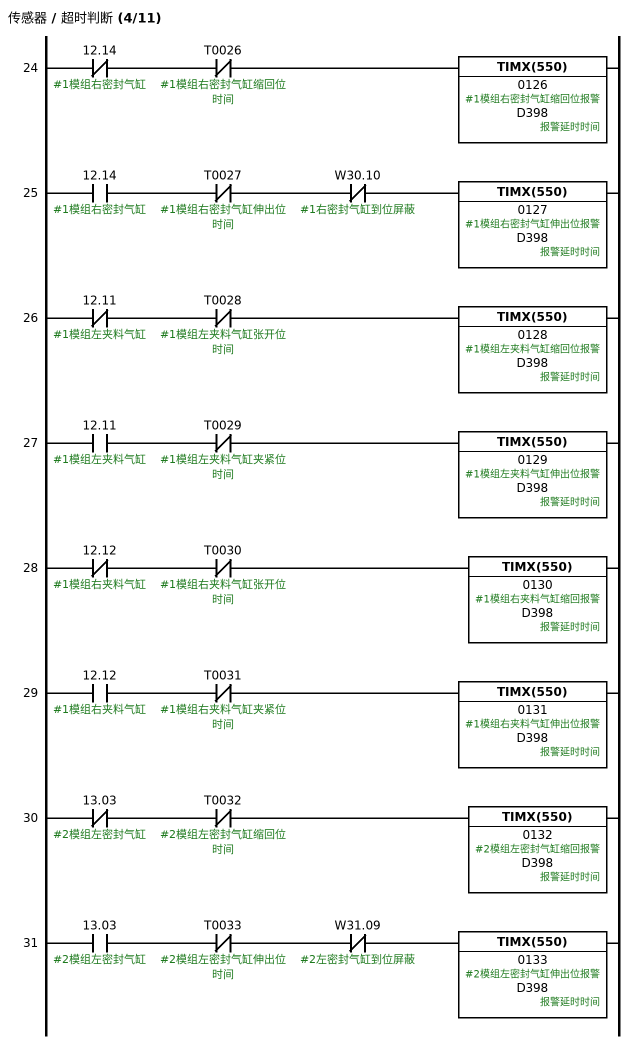
; [picture p65: 传感器 / 超时判断, rungs 24-31]
; rung 24
LDNOT 12.14  ; #1模组右密封气缸
ANDNOT T0026  ; #1模组右密封气缸缩回位时间
TIMX(550) 0126 D398  ; 报警延时时间, #1模组右密封气缸缩回位报警
; rung 25
LD 12.14  ; #1模组右密封气缸
ANDNOT T0027  ; #1模组右密封气缸伸出位时间
ANDNOT W30.10  ; #1右密封气缸到位屏蔽
TIMX(550) 0127 D398  ; 报警延时时间, #1模组右密封气缸伸出位报警
; rung 26
LDNOT 12.11  ; #1模组左夹料气缸
ANDNOT T0028  ; #1模组左夹料气缸张开位时间
TIMX(550) 0128 D398  ; 报警延时时间, #1模组左夹料气缸缩回位报警
; rung 27
LD 12.11  ; #1模组左夹料气缸
ANDNOT T0029  ; #1模组左夹料气缸夹紧位时间
TIMX(550) 0129 D398  ; 报警延时时间, #1模组左夹料气缸伸出位报警
; rung 28
LDNOT 12.12  ; #1模组右夹料气缸
ANDNOT T0030  ; #1模组右夹料气缸张开位时间
TIMX(550) 0130 D398  ; 报警延时时间, #1模组右夹料气缸缩回报警
; rung 29
LD 12.12  ; #1模组右夹料气缸
ANDNOT T0031  ; #1模组右夹料气缸夹紧位时间
TIMX(550) 0131 D398  ; 报警延时时间, #1模组右夹料气缸伸出位报警
; rung 30
LDNOT 13.03  ; #2模组左密封气缸
ANDNOT T0032  ; #2模组左密封气缸缩回位时间
TIMX(550) 0132 D398  ; 报警延时时间, #2模组左密封气缸缩回报警
; rung 31
LD 13.03  ; #2模组左密封气缸
ANDNOT T0033  ; #2模组左密封气缸伸出位时间
ANDNOT W31.09  ; #2左密封气缸到位屏蔽
TIMX(550) 0133 D398  ; 报警延时时间, #2模组左密封气缸伸出位报警

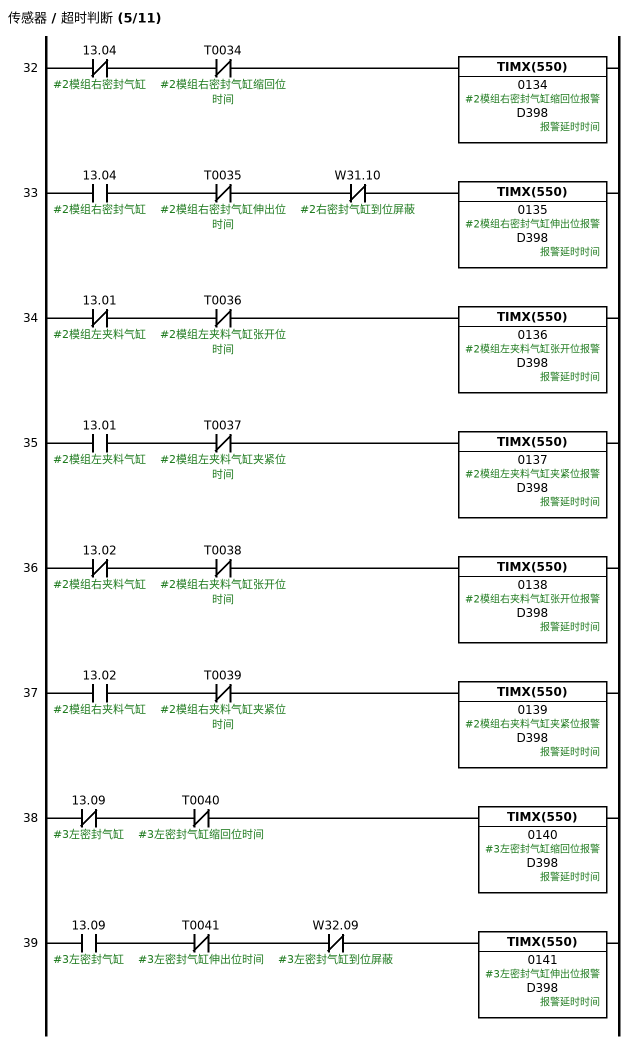
; rung 32
LDNOT 13.04  ; #2模组右密封气缸
ANDNOT T0034  ; #2模组右密封气缸缩回位时间
TIMX(550) 0134 D398  ; 报警延时时间, #2模组右密封气缸缩回位报警
; rung 33
LD 13.04  ; #2模组右密封气缸
ANDNOT T0035  ; #2模组右密封气缸伸出位时间
ANDNOT W31.10  ; #2右密封气缸到位屏蔽
TIMX(550) 0135 D398  ; 报警延时时间, #2模组右密封气缸伸出位报警
; rung 34
LDNOT 13.01  ; #2模组左夹料气缸
ANDNOT T0036  ; #2模组左夹料气缸张开位时间
TIMX(550) 0136 D398  ; 报警延时时间, #2模组左夹料气缸张开位报警
; rung 35
LD 13.01  ; #2模组左夹料气缸
ANDNOT T0037  ; #2模组左夹料气缸夹紧位时间
TIMX(550) 0137 D398  ; 报警延时时间, #2模组左夹料气缸夹紧位报警
; rung 36
LDNOT 13.02  ; #2模组右夹料气缸
ANDNOT T0038  ; #2模组右夹料气缸张开位时间
TIMX(550) 0138 D398  ; 报警延时时间, #2模组右夹料气缸张开位报警
; rung 37
LD 13.02  ; #2模组右夹料气缸
ANDNOT T0039  ; #2模组右夹料气缸夹紧位时间
TIMX(550) 0139 D398  ; 报警延时时间, #2模组右夹料气缸夹紧位报警
; rung 38
LDNOT 13.09  ; #3左密封气缸
ANDNOT T0040  ; #3左密封气缸缩回位时间
TIMX(550) 0140 D398  ; 报警延时时间, #3左密封气缸缩回位报警
; rung 39
LD 13.09  ; #3左密封气缸
ANDNOT T0041  ; #3左密封气缸伸出位时间
ANDNOT W32.09  ; #3左密封气缸到位屏蔽
TIMX(550) 0141 D398  ; 报警延时时间, #3左密封气缸伸出位报警

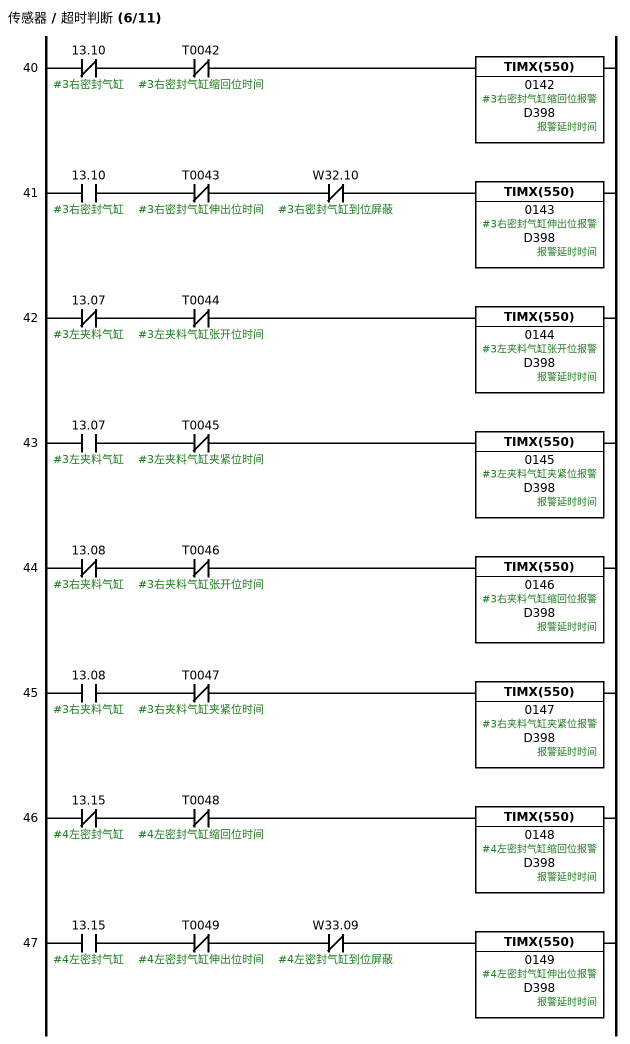
; rung 40
LDNOT 13.10  ; #3右密封气缸
ANDNOT T0042  ; #3右密封气缸缩回位时间
TIMX(550) 0142 D398  ; 报警延时时间, #3右密封气缸缩回位报警
; rung 41
LD 13.10  ; #3右密封气缸
ANDNOT T0043  ; #3右密封气缸伸出位时间
ANDNOT W32.10  ; #3右密封气缸到位屏蔽
TIMX(550) 0143 D398  ; 报警延时时间, #3右密封气缸伸出位报警
; rung 42
LDNOT 13.07  ; #3左夹料气缸
ANDNOT T0044  ; #3左夹料气缸张开位时间
TIMX(550) 0144 D398  ; 报警延时时间, #3左夹料气缸张开位报警
; rung 43
LD 13.07  ; #3左夹料气缸
ANDNOT T0045  ; #3左夹料气缸夹紧位时间
TIMX(550) 0145 D398  ; 报警延时时间, #3左夹料气缸夹紧位报警
; rung 44
LDNOT 13.08  ; #3右夹料气缸
ANDNOT T0046  ; #3右夹料气缸张开位时间
TIMX(550) 0146 D398  ; 报警延时时间, #3右夹料气缸缩回位报警
; rung 45
LD 13.08  ; #3右夹料气缸
ANDNOT T0047  ; #3右夹料气缸夹紧位时间
TIMX(550) 0147 D398  ; 报警延时时间, #3右夹料气缸夹紧位报警
; rung 46
LDNOT 13.15  ; #4左密封气缸
ANDNOT T0048  ; #4左密封气缸缩回位时间
TIMX(550) 0148 D398  ; 报警延时时间, #4左密封气缸缩回位报警
; rung 47
LD 13.15  ; #4左密封气缸
ANDNOT T0049  ; #4左密封气缸伸出位时间
ANDNOT W33.09  ; #4左密封气缸到位屏蔽
TIMX(550) 0149 D398  ; 报警延时时间, #4左密封气缸伸出位报警

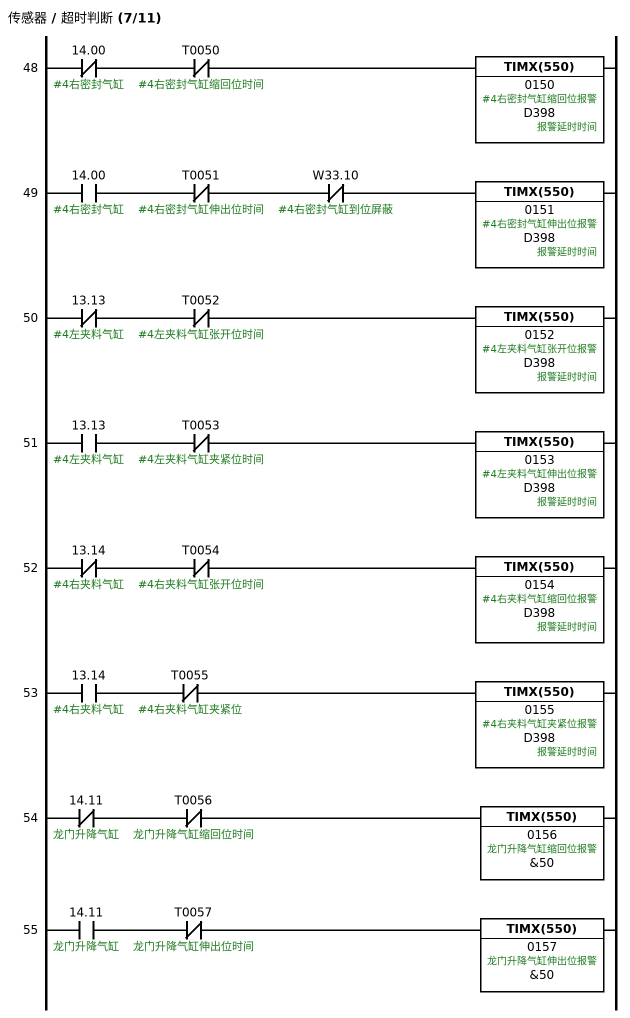
; rung 48
LDNOT 14.00  ; #4右密封气缸
ANDNOT T0050  ; #4右密封气缸缩回位时间
TIMX(550) 0150 D398  ; 报警延时时间, #4右密封气缸缩回位报警
; rung 49
LD 14.00  ; #4右密封气缸
ANDNOT T0051  ; #4右密封气缸伸出位时间
ANDNOT W33.10  ; #4右密封气缸到位屏蔽
TIMX(550) 0151 D398  ; 报警延时时间, #4右密封气缸伸出位报警
; rung 50
LDNOT 13.13  ; #4左夹料气缸
ANDNOT T0052  ; #4左夹料气缸张开位时间
TIMX(550) 0152 D398  ; 报警延时时间, #4左夹料气缸张开位报警
; rung 51
LD 13.13  ; #4左夹料气缸
ANDNOT T0053  ; #4左夹料气缸夹紧位时间
TIMX(550) 0153 D398  ; 报警延时时间, #4左夹料气缸伸出位报警
; rung 52
LDNOT 13.14  ; #4右夹料气缸
ANDNOT T0054  ; #4右夹料气缸张开位时间
TIMX(550) 0154 D398  ; 报警延时时间, #4右夹料气缸缩回位报警
; rung 53
LD 13.14  ; #4右夹料气缸
ANDNOT T0055  ; #4右夹料气缸夹紧位
TIMX(550) 0155 D398  ; 报警延时时间, #4右夹料气缸夹紧位报警
; rung 54
LDNOT 14.11  ; 龙门升降气缸
ANDNOT T0056  ; 龙门升降气缸缩回位时间
TIMX(550) 0156 &50  ; 龙门升降气缸缩回位报警
; rung 55
LD 14.11  ; 龙门升降气缸
ANDNOT T0057  ; 龙门升降气缸伸出位时间
TIMX(550) 0157 &50  ; 龙门升降气缸伸出位报警

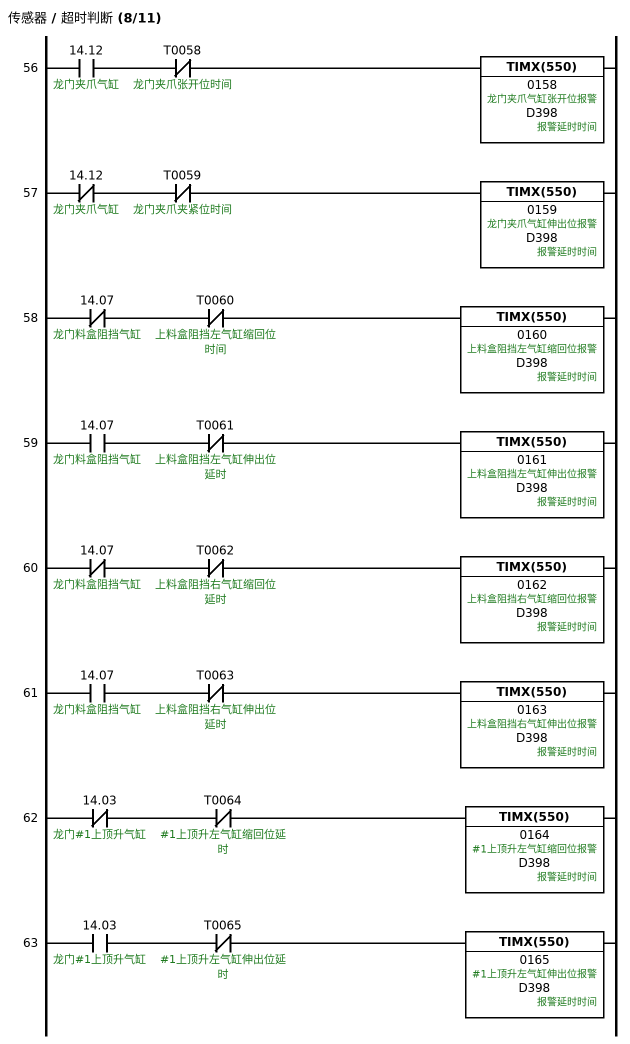
; rung 56
LD 14.12  ; 龙门夹爪气缸
ANDNOT T0058  ; 龙门夹爪张开位时间
TIMX(550) 0158 D398  ; 报警延时时间, 龙门夹爪气缸张开位报警
; rung 57
LDNOT 14.12  ; 龙门夹爪气缸
ANDNOT T0059  ; 龙门夹爪夹紧位时间
TIMX(550) 0159 D398  ; 报警延时时间, 龙门夹爪气缸伸出位报警
; rung 58
LDNOT 14.07  ; 龙门料盒阻挡气缸
ANDNOT T0060  ; 上料盒阻挡左气缸缩回位时间
TIMX(550) 0160 D398  ; 报警延时时间, 上料盒阻挡左气缸缩回位报警
; rung 59
LD 14.07  ; 龙门料盒阻挡气缸
ANDNOT T0061  ; 上料盒阻挡左气缸伸出位延时
TIMX(550) 0161 D398  ; 报警延时时间, 上料盒阻挡左气缸伸出位报警
; rung 60
LDNOT 14.07  ; 龙门料盒阻挡气缸
ANDNOT T0062  ; 上料盒阻挡右气缸缩回位延时
TIMX(550) 0162 D398  ; 报警延时时间, 上料盒阻挡右气缸缩回位报警
; rung 61
LD 14.07  ; 龙门料盒阻挡气缸
ANDNOT T0063  ; 上料盒阻挡右气缸伸出位延时
TIMX(550) 0163 D398  ; 报警延时时间, 上料盒阻挡右气缸伸出位报警
; rung 62
LDNOT 14.03  ; 龙门#1上顶升气缸
ANDNOT T0064  ; #1上顶升左气缸缩回位延时
TIMX(550) 0164 D398  ; 报警延时时间, #1上顶升左气缸缩回位报警
; rung 63
LD 14.03  ; 龙门#1上顶升气缸
ANDNOT T0065  ; #1上顶升左气缸伸出位延时
TIMX(550) 0165 D398  ; 报警延时时间, #1上顶升左气缸伸出位报警

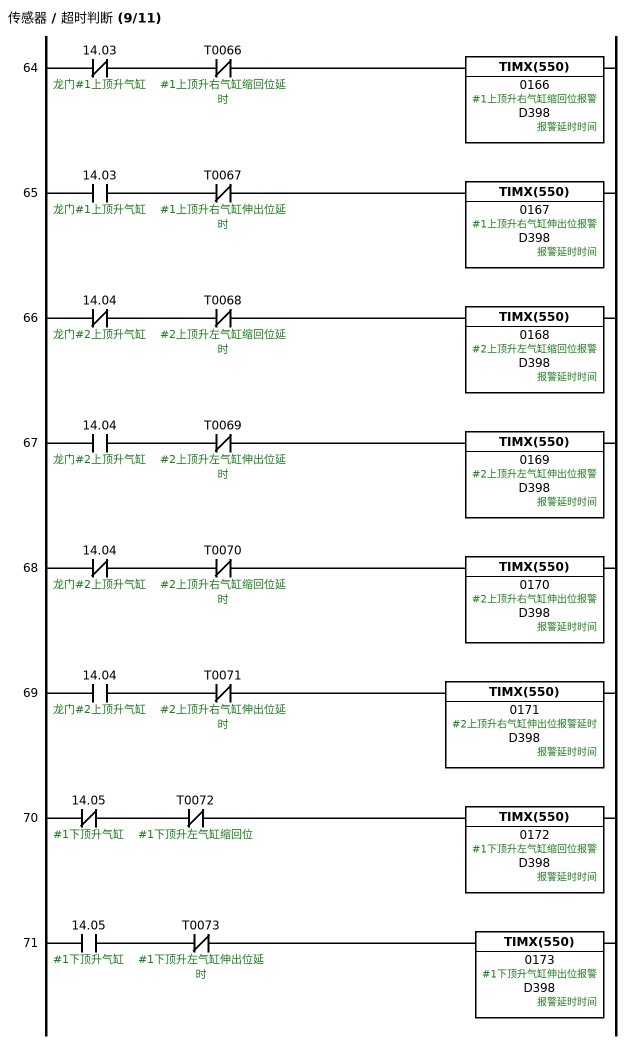
; rung 64
LDNOT 14.03  ; 龙门#1上顶升气缸
ANDNOT T0066  ; #1上顶升右气缸缩回位延时
TIMX(550) 0166 D398  ; 报警延时时间, #1上顶升右气缸缩回位报警
; rung 65
LD 14.03  ; 龙门#1上顶升气缸
ANDNOT T0067  ; #1上顶升右气缸伸出位延时
TIMX(550) 0167 D398  ; 报警延时时间, #1上顶升右气缸伸出位报警
; rung 66
LDNOT 14.04  ; 龙门#2上顶升气缸
ANDNOT T0068  ; #2上顶升左气缸缩回位延时
TIMX(550) 0168 D398  ; 报警延时时间, #2上顶升左气缸缩回位报警
; rung 67
LD 14.04  ; 龙门#2上顶升气缸
ANDNOT T0069  ; #2上顶升左气缸伸出位延时
TIMX(550) 0169 D398  ; 报警延时时间, #2上顶升左气缸伸出位报警
; rung 68
LDNOT 14.04  ; 龙门#2上顶升气缸
ANDNOT T0070  ; #2上顶升右气缸缩回位延时
TIMX(550) 0170 D398  ; 报警延时时间, #2上顶升右气缸伸出位报警
; rung 69
LD 14.04  ; 龙门#2上顶升气缸
ANDNOT T0071  ; #2上顶升右气缸伸出位延时
TIMX(550) 0171 D398  ; 报警延时时间, #2上顶升右气缸伸出位报警延时
; rung 70
LDNOT 14.05  ; #1下顶升气缸
ANDNOT T0072  ; #1下顶升左气缸缩回位
TIMX(550) 0172 D398  ; 报警延时时间, #1下顶升左气缸缩回位报警
; rung 71
LD 14.05  ; #1下顶升气缸
ANDNOT T0073  ; #1下顶升左气缸伸出位延时
TIMX(550) 0173 D398  ; 报警延时时间, #1下顶升气缸伸出位报警

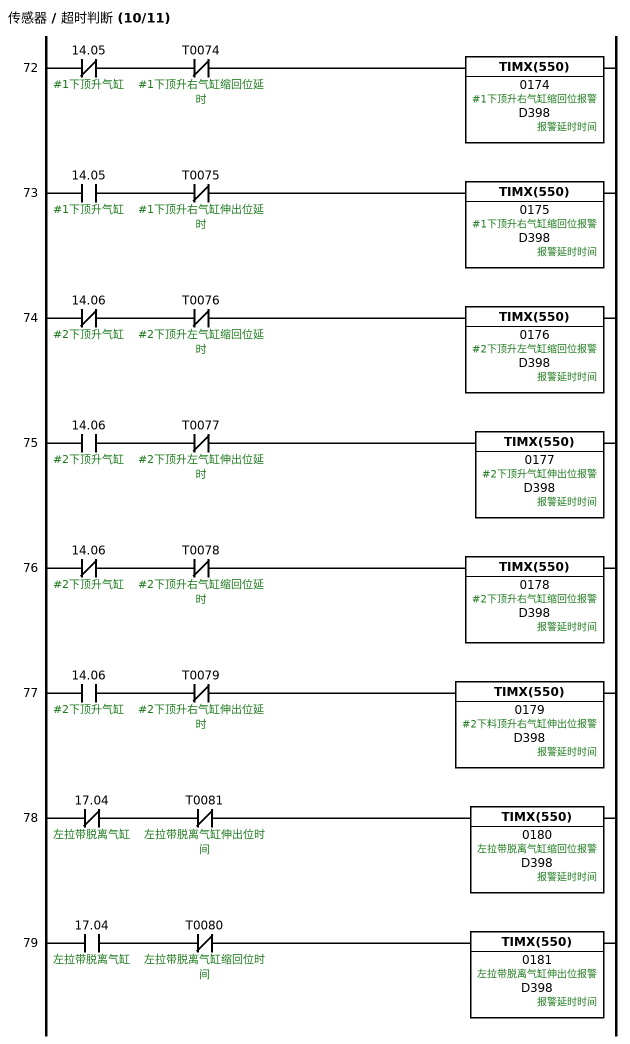
; rung 72
LDNOT 14.05  ; #1下顶升气缸
ANDNOT T0074  ; #1下顶升右气缸缩回位延时
TIMX(550) 0174 D398  ; 报警延时时间, #1下顶升右气缸缩回位报警
; rung 73
LD 14.05  ; #1下顶升气缸
ANDNOT T0075  ; #1下顶升右气缸伸出位延时
TIMX(550) 0175 D398  ; 报警延时时间, #1下顶升右气缸缩回位报警
; rung 74
LDNOT 14.06  ; #2下顶升气缸
ANDNOT T0076  ; #2下顶升左气缸缩回位延时
TIMX(550) 0176 D398  ; 报警延时时间, #2下顶升左气缸缩回位报警
; rung 75
LD 14.06  ; #2下顶升气缸
ANDNOT T0077  ; #2下顶升左气缸伸出位延时
TIMX(550) 0177 D398  ; 报警延时时间, #2下顶升气缸伸出位报警
; rung 76
LDNOT 14.06  ; #2下顶升气缸
ANDNOT T0078  ; #2下顶升右气缸缩回位延时
TIMX(550) 0178 D398  ; 报警延时时间, #2下顶升右气缸缩回位报警
; rung 77
LD 14.06  ; #2下顶升气缸
ANDNOT T0079  ; #2下顶升右气缸伸出位延时
TIMX(550) 0179 D398  ; 报警延时时间, #2下料顶升右气缸伸出位报警
; rung 78
LDNOT 17.04  ; 左拉带脱离气缸
ANDNOT T0081  ; 左拉带脱离气缸伸出位时间
TIMX(550) 0180 D398  ; 报警延时时间, 左拉带脱离气缸缩回位报警
; rung 79
LD 17.04  ; 左拉带脱离气缸
ANDNOT T0080  ; 左拉带脱离气缸缩回位时间
TIMX(550) 0181 D398  ; 报警延时时间, 左拉带脱离气缸伸出位报警

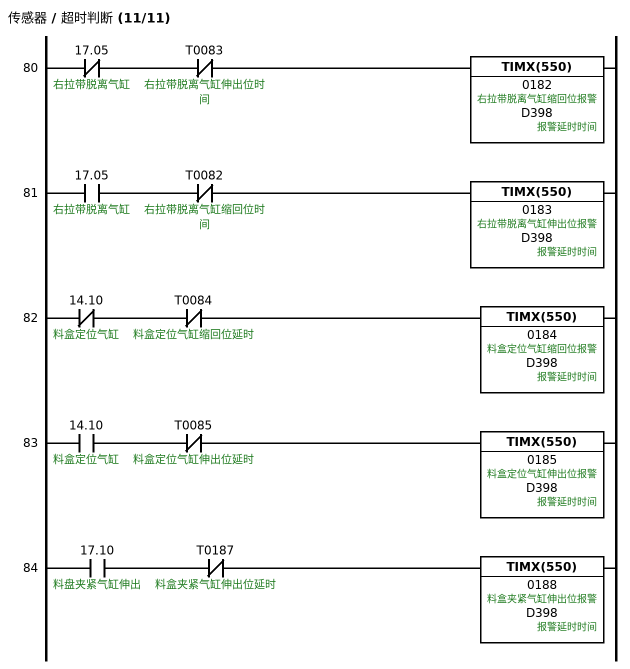
; rung 80
LDNOT 17.05  ; 右拉带脱离气缸
ANDNOT T0083  ; 右拉带脱离气缸伸出位时间
TIMX(550) 0182 D398  ; 报警延时时间, 右拉带脱离气缸缩回位报警
; rung 81
LD 17.05  ; 右拉带脱离气缸
ANDNOT T0082  ; 右拉带脱离气缸缩回位时间
TIMX(550) 0183 D398  ; 报警延时时间, 右拉带脱离气缸伸出位报警
; rung 82
LDNOT 14.10  ; 料盒定位气缸
ANDNOT T0084  ; 料盒定位气缸缩回位延时
TIMX(550) 0184 D398  ; 报警延时时间, 料盒定位气缸缩回位报警
; rung 83
LD 14.10  ; 料盒定位气缸
ANDNOT T0085  ; 料盒定位气缸伸出位延时
TIMX(550) 0185 D398  ; 报警延时时间, 料盒定位气缸伸出位报警
; rung 84
LD 17.10  ; 料盘夹紧气缸伸出
ANDNOT T0187  ; 料盒夹紧气缸伸出位延时
TIMX(550) 0188 D398  ; 报警延时时间, 料盒夹紧气缸伸出位报警

### Section END
; rung 0
END(001)

## Program 上料机构 (cyclic task 2)

### Section 扫码，检测手动

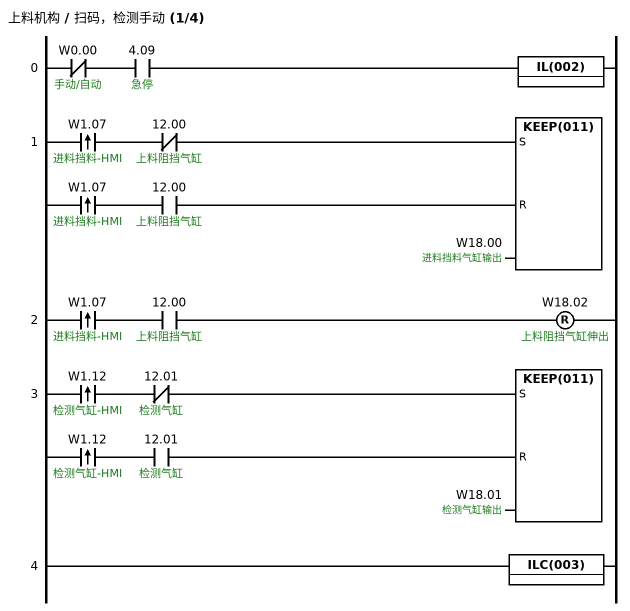
; rung 0
LDNOT W0.00  ; 手动/自动
AND 4.09  ; 急停
IL(002)
; rung 1
@LD W1.07  ; 进料挡料-HMI
ANDNOT 12.00  ; 上料阻挡气缸
@LD W1.07  ; 进料挡料-HMI
AND 12.00  ; 上料阻挡气缸
KEEP(011) W18.00  ; 进料挡料气缸输出
; rung 2
@LD W1.07  ; 进料挡料-HMI
AND 12.00  ; 上料阻挡气缸
RSET W18.02  ; 上料阻挡气缸伸出
; rung 3
@LD W1.12  ; 检测气缸-HMI
ANDNOT 12.01  ; 检测气缸
@LD W1.12  ; 检测气缸-HMI
AND 12.01  ; 检测气缸
KEEP(011) W18.01  ; 检测气缸输出
; rung 4
ILC(003)

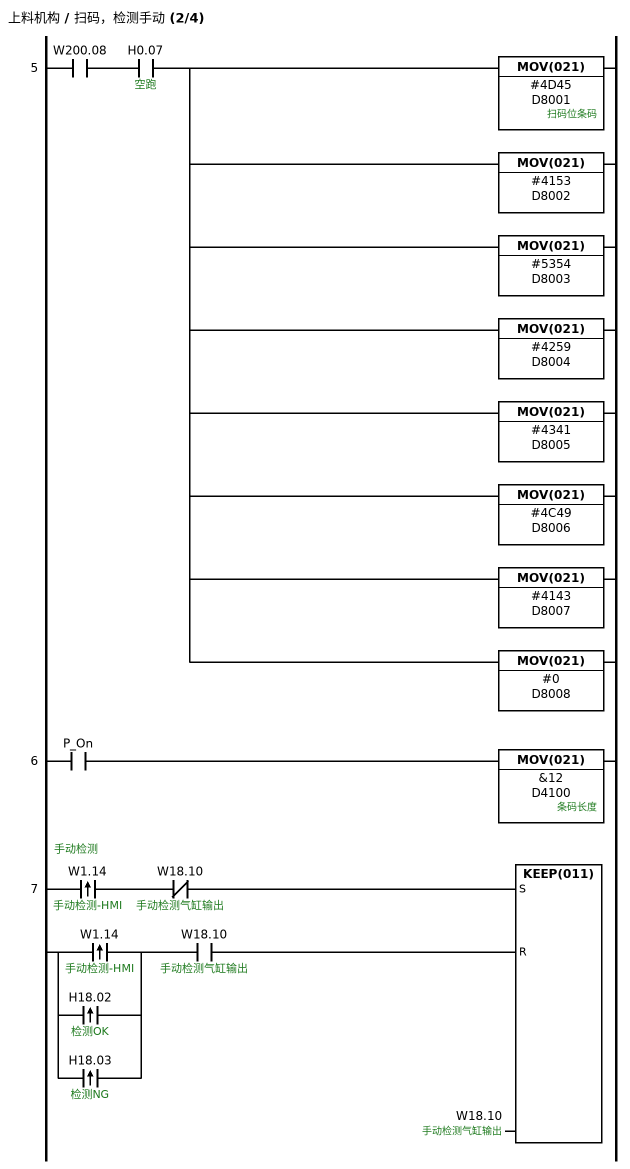
; rung 5
LD W200.08
AND H0.07  ; 空跑
MOV(021) #4D45 D8001  ; 扫码位条码
MOV(021) #4153 D8002
MOV(021) #5354 D8003
MOV(021) #4259 D8004
MOV(021) #4341 D8005
MOV(021) #4C49 D8006
MOV(021) #4143 D8007
MOV(021) #0 D8008
; rung 6
LD P_On
MOV(021) &12 D4100  ; 条码长度
; rung 7: 手动检测
@LD W1.14  ; 手动检测-HMI
ANDNOT W18.10  ; 手动检测气缸输出
@LD W1.14  ; 手动检测-HMI
@OR H18.02  ; 检测OK
@OR H18.03  ; 检测NG
AND W18.10  ; 手动检测气缸输出
KEEP(011) W18.10  ; 手动检测气缸输出

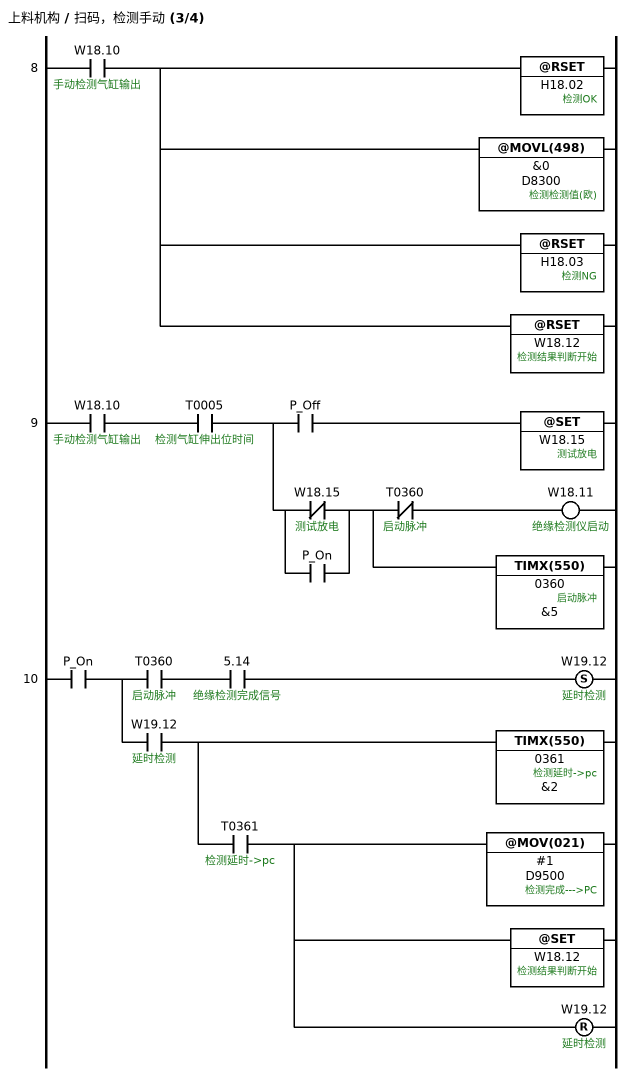
; rung 8
LD W18.10  ; 手动检测气缸输出
@RSET H18.02  ; 检测OK
@MOVL(498) &0 D8300  ; 检测检测值(欧)
@RSET H18.03  ; 检测NG
@RSET W18.12  ; 检测结果判断开始
; rung 9
LD W18.10  ; 手动检测气缸输出
AND T0005  ; 检测气缸伸出位时间
OUT TR0
AND P_Off
@SET W18.15  ; 测试放电
LD TR0
LDNOT W18.15  ; 测试放电
OR P_On
ANDLD
OUT TR0
ANDNOT T0360  ; 启动脉冲
OUT W18.11  ; 绝缘检测仪启动
LD TR0
TIMX(550) 0360 &5  ; 启动脉冲
; rung 10
LD P_On
OUT TR0
AND T0360  ; 启动脉冲
AND 5.14  ; 绝缘检测完成信号
SET W19.12  ; 延时检测
LD TR0
AND W19.12  ; 延时检测
TIMX(550) 0361 &2  ; 检测延时->pc
AND T0361  ; 检测延时->pc
@MOV(021) #1 D9500  ; 检测完成--->PC
@SET W18.12  ; 检测结果判断开始
RSET W19.12  ; 延时检测

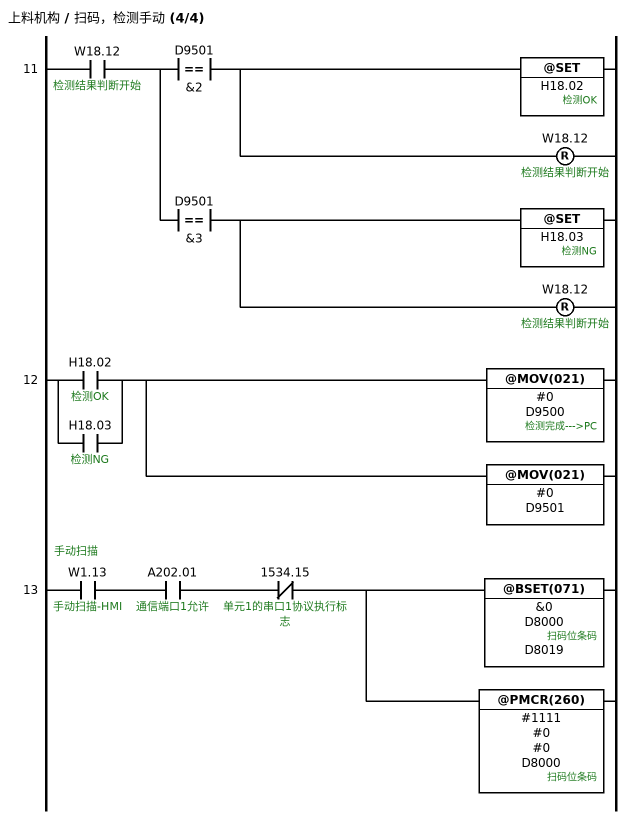
; rung 11
LD W18.12  ; 检测结果判断开始
OUT TR0
AND=(300) D9501 &2
@SET H18.02  ; 检测OK
RSET W18.12  ; 检测结果判断开始
LD TR0
AND=(300) D9501 &3
@SET H18.03  ; 检测NG
RSET W18.12  ; 检测结果判断开始
; rung 12
LD H18.02  ; 检测OK
OR H18.03  ; 检测NG
@MOV(021) #0 D9500  ; 检测完成--->PC
@MOV(021) #0 D9501
; rung 13: 手动扫描
LD W1.13  ; 手动扫描-HMI
AND A202.01  ; 通信端口1允许
ANDNOT 1534.15  ; 单元1的串口1协议执行标志
@BSET(071) &0 D8000 D8019  ; 扫码位条码
@PMCR(260) #1111 #0 #0 D8000  ; 扫码位条码

### Section 扫码，检测自动

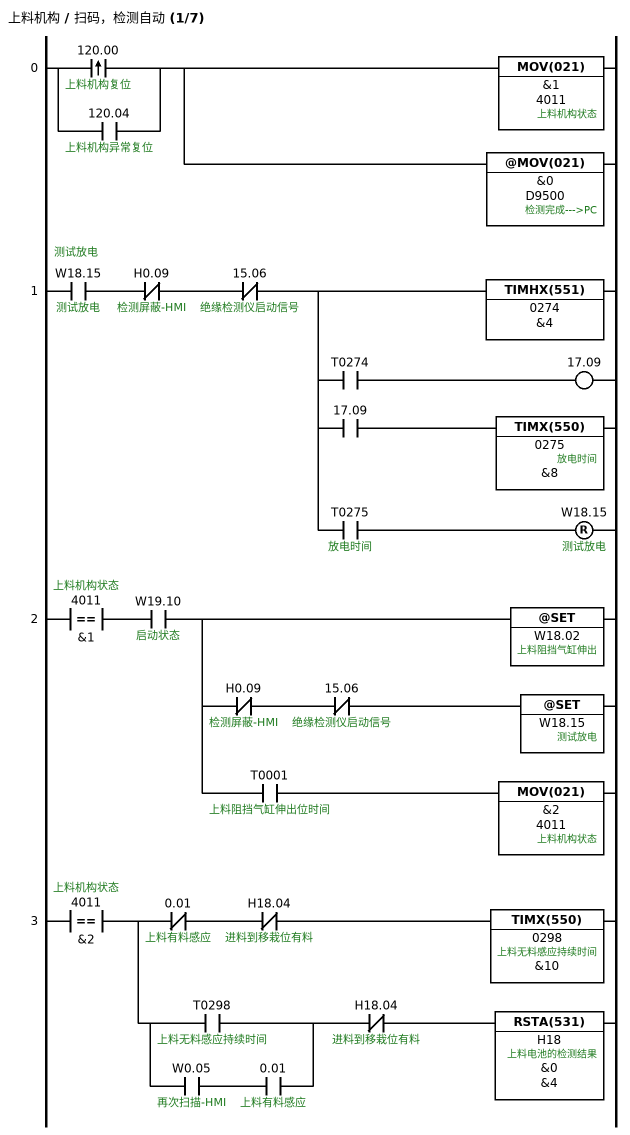
; rung 0
@LD 120.00  ; 上料机构复位
OR 120.04  ; 上料机构异常复位
MOV(021) &1 4011  ; 上料机构状态
@MOV(021) &0 D9500  ; 检测完成--->PC
; rung 1: 测试放电
LD W18.15  ; 测试放电
ANDNOT H0.09  ; 检测屏蔽-HMI
ANDNOT 15.06  ; 绝缘检测仪启动信号
OUT TR0
TIMHX(551) 0274 &4
AND T0274
OUT 17.09
LD TR0
AND 17.09
TIMX(550) 0275 &8  ; 放电时间
LD TR0
AND T0275  ; 放电时间
RSET W18.15  ; 测试放电
; rung 2
LD=(300) 4011 &1  ; 上料机构状态
AND W19.10  ; 启动状态
OUT TR0
@SET W18.02  ; 上料阻挡气缸伸出
ANDNOT H0.09  ; 检测屏蔽-HMI
ANDNOT 15.06  ; 绝缘检测仪启动信号
@SET W18.15  ; 测试放电
LD TR0
AND T0001  ; 上料阻挡气缸伸出位时间
MOV(021) &2 4011  ; 上料机构状态
; rung 3
LD=(300) 4011 &2  ; 上料机构状态
OUT TR0
ANDNOT 0.01  ; 上料有料感应
ANDNOT H18.04  ; 进料到移栽位有料
TIMX(550) 0298 &10  ; 上料无料感应持续时间
LD TR0
LD T0298  ; 上料无料感应持续时间
LD W0.05  ; 再次扫描-HMI
AND 0.01  ; 上料有料感应
ORLD
ANDLD
ANDNOT H18.04  ; 进料到移栽位有料
RSTA(531) H18 &0 &4  ; 上料电池的检测结果

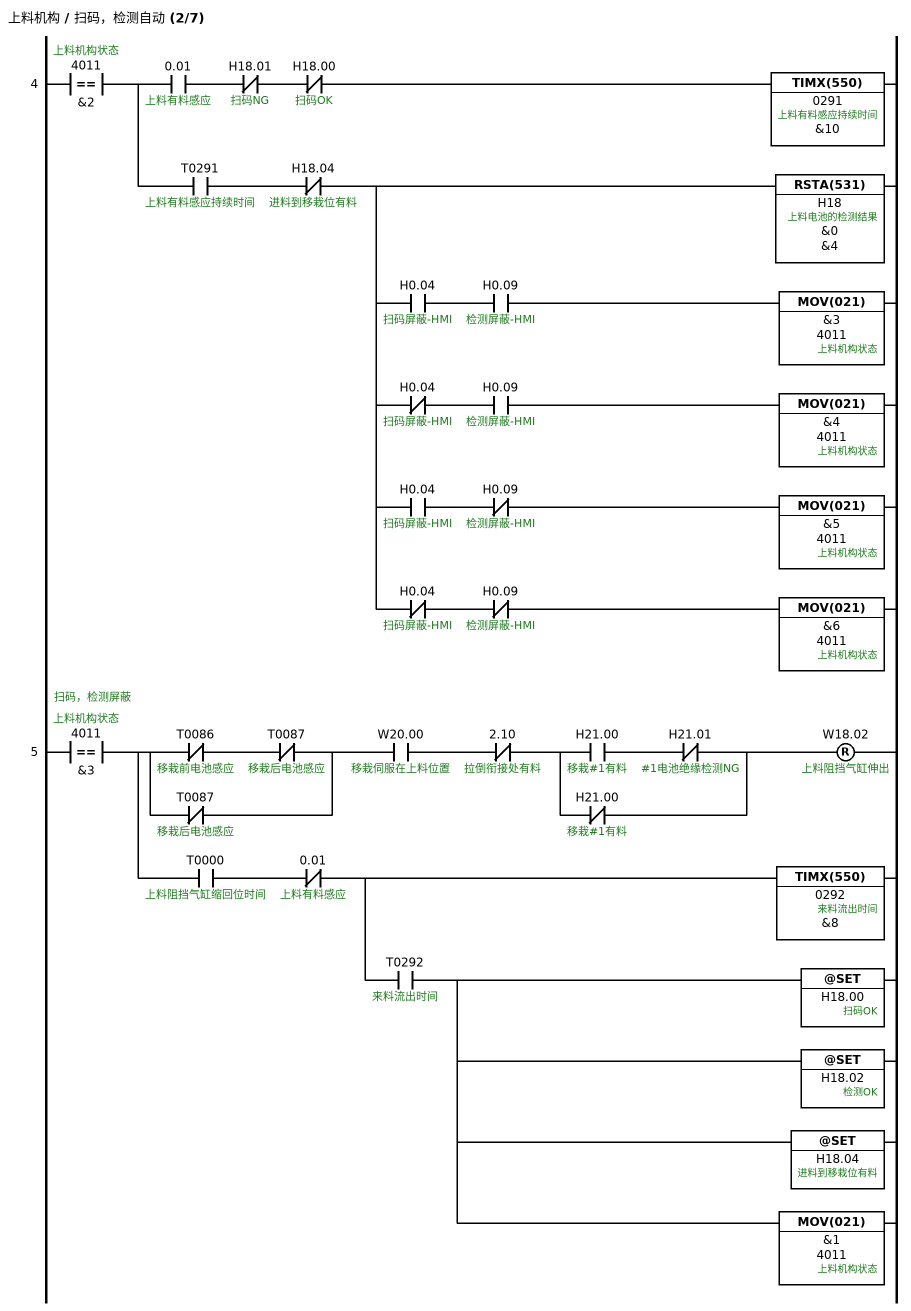
; rung 4
LD=(300) 4011 &2  ; 上料机构状态
OUT TR0
AND 0.01  ; 上料有料感应
ANDNOT H18.01  ; 扫码NG
ANDNOT H18.00  ; 扫码OK
TIMX(550) 0291 &10  ; 上料有料感应持续时间
LD TR0
AND T0291  ; 上料有料感应持续时间
ANDNOT H18.04  ; 进料到移栽位有料
OUT TR0
RSTA(531) H18 &0 &4  ; 上料电池的检测结果
AND H0.04  ; 扫码屏蔽-HMI
AND H0.09  ; 检测屏蔽-HMI
MOV(021) &3 4011  ; 上料机构状态
LD TR0
ANDNOT H0.04  ; 扫码屏蔽-HMI
AND H0.09  ; 检测屏蔽-HMI
MOV(021) &4 4011  ; 上料机构状态
LD TR0
AND H0.04  ; 扫码屏蔽-HMI
ANDNOT H0.09  ; 检测屏蔽-HMI
MOV(021) &5 4011  ; 上料机构状态
LD TR0
ANDNOT H0.04  ; 扫码屏蔽-HMI
ANDNOT H0.09  ; 检测屏蔽-HMI
MOV(021) &6 4011  ; 上料机构状态
; rung 5: 扫码，检测屏蔽
LD=(300) 4011 &3  ; 上料机构状态
OUT TR0
LDNOT T0086  ; 移栽前电池感应
ANDNOT T0087  ; 移栽后电池感应
ORNOT T0087  ; 移栽后电池感应
ANDLD
AND W20.00  ; 移栽伺服在上料位置
ANDNOT 2.10  ; 拉倒衔接处有料
LD H21.00  ; 移栽#1有料
ANDNOT H21.01  ; #1电池绝缘检测NG
ORNOT H21.00  ; 移栽#1有料
ANDLD
RSET W18.02  ; 上料阻挡气缸伸出
LD TR0
AND T0000  ; 上料阻挡气缸缩回位时间
ANDNOT 0.01  ; 上料有料感应
TIMX(550) 0292 &8  ; 来料流出时间
AND T0292  ; 来料流出时间
@SET H18.00  ; 扫码OK
@SET H18.02  ; 检测OK
@SET H18.04  ; 进料到移栽位有料
MOV(021) &1 4011  ; 上料机构状态

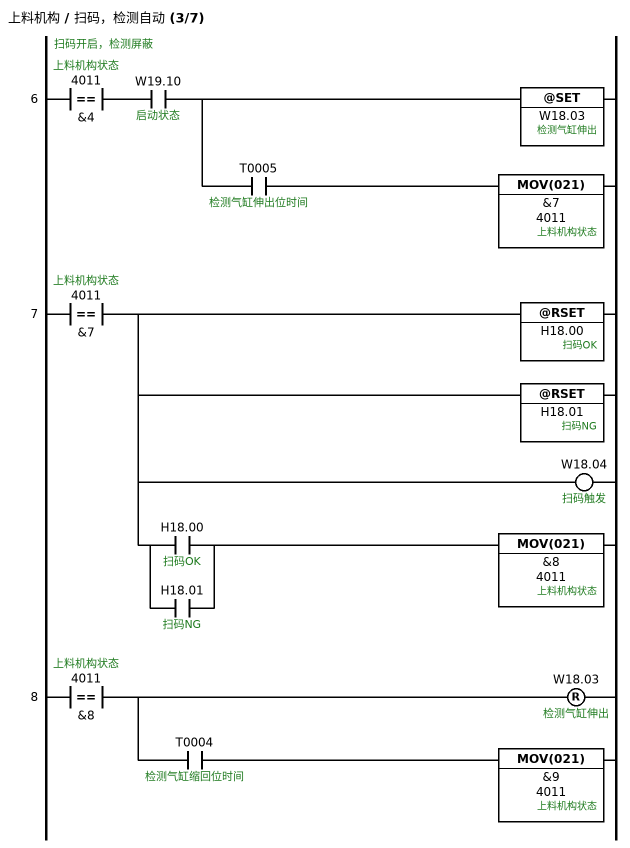
; rung 6: 扫码开启，检测屏蔽
LD=(300) 4011 &4  ; 上料机构状态
AND W19.10  ; 启动状态
@SET W18.03  ; 检测气缸伸出
AND T0005  ; 检测气缸伸出位时间
MOV(021) &7 4011  ; 上料机构状态
; rung 7
LD=(300) 4011 &7  ; 上料机构状态
@RSET H18.00  ; 扫码OK
@RSET H18.01  ; 扫码NG
OUT W18.04  ; 扫码触发
LD H18.00  ; 扫码OK
OR H18.01  ; 扫码NG
ANDLD
MOV(021) &8 4011  ; 上料机构状态
; rung 8
LD=(300) 4011 &8  ; 上料机构状态
RSET W18.03  ; 检测气缸伸出
AND T0004  ; 检测气缸缩回位时间
MOV(021) &9 4011  ; 上料机构状态

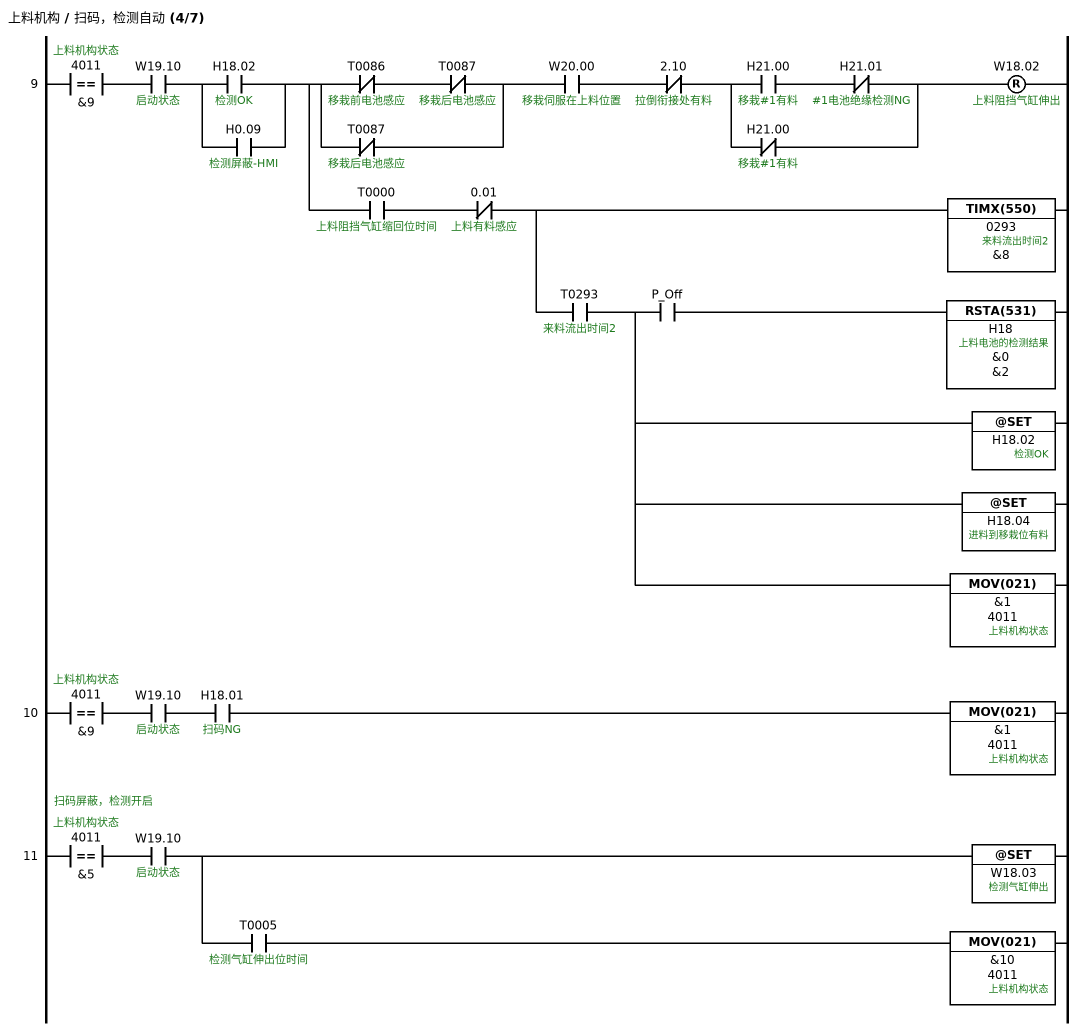
; rung 9
LD=(300) 4011 &9  ; 上料机构状态
AND W19.10  ; 启动状态
LD H18.02  ; 检测OK
OR H0.09  ; 检测屏蔽-HMI
ANDLD
OUT TR0
LDNOT T0086  ; 移栽前电池感应
ANDNOT T0087  ; 移栽后电池感应
ORNOT T0087  ; 移栽后电池感应
ANDLD
AND W20.00  ; 移栽伺服在上料位置
ANDNOT 2.10  ; 拉倒衔接处有料
LD H21.00  ; 移栽#1有料
ANDNOT H21.01  ; #1电池绝缘检测NG
ORNOT H21.00  ; 移栽#1有料
ANDLD
RSET W18.02  ; 上料阻挡气缸伸出
LD TR0
AND T0000  ; 上料阻挡气缸缩回位时间
ANDNOT 0.01  ; 上料有料感应
TIMX(550) 0293 &8  ; 来料流出时间2
AND T0293  ; 来料流出时间2
OUT TR0
AND P_Off
RSTA(531) H18 &0 &2  ; 上料电池的检测结果
LD TR0
@SET H18.02  ; 检测OK
@SET H18.04  ; 进料到移栽位有料
MOV(021) &1 4011  ; 上料机构状态
; rung 10
LD=(300) 4011 &9  ; 上料机构状态
AND W19.10  ; 启动状态
AND H18.01  ; 扫码NG
MOV(021) &1 4011  ; 上料机构状态
; rung 11: 扫码屏蔽，检测开启
LD=(300) 4011 &5  ; 上料机构状态
AND W19.10  ; 启动状态
@SET W18.03  ; 检测气缸伸出
AND T0005  ; 检测气缸伸出位时间
MOV(021) &10 4011  ; 上料机构状态

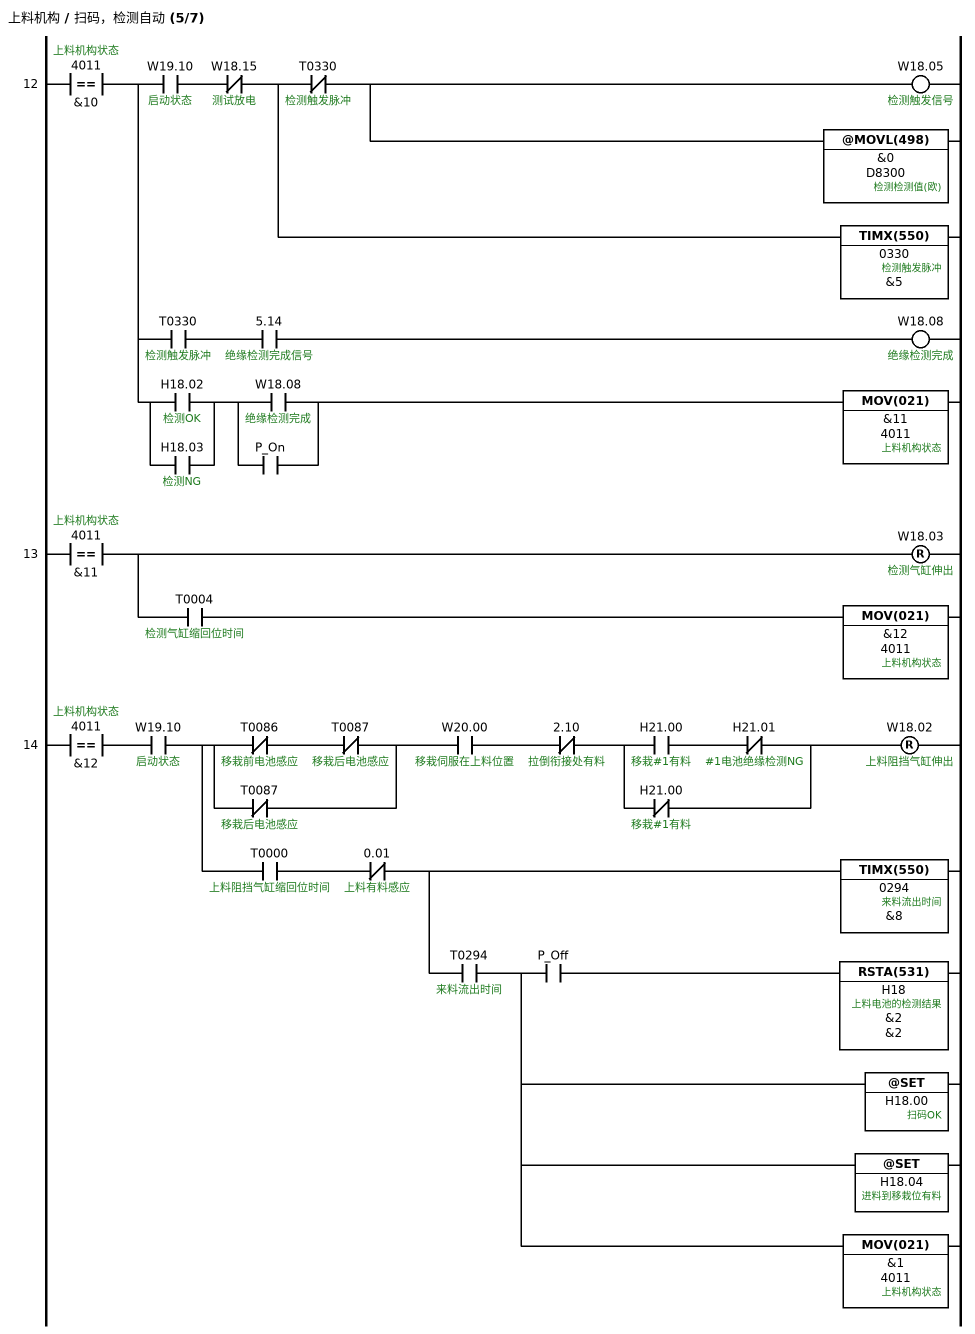
; rung 12
LD=(300) 4011 &10  ; 上料机构状态
OUT TR0
AND W19.10  ; 启动状态
ANDNOT W18.15  ; 测试放电
OUT TR1
ANDNOT T0330  ; 检测触发脉冲
OUT W18.05  ; 检测触发信号
@MOVL(498) &0 D8300  ; 检测检测值(欧)
LD TR1
TIMX(550) 0330 &5  ; 检测触发脉冲
LD TR0
AND T0330  ; 检测触发脉冲
AND 5.14  ; 绝缘检测完成信号
OUT W18.08  ; 绝缘检测完成
LD TR0
LD H18.02  ; 检测OK
OR H18.03  ; 检测NG
ANDLD
LD W18.08  ; 绝缘检测完成
OR P_On
ANDLD
MOV(021) &11 4011  ; 上料机构状态
; rung 13
LD=(300) 4011 &11  ; 上料机构状态
RSET W18.03  ; 检测气缸伸出
AND T0004  ; 检测气缸缩回位时间
MOV(021) &12 4011  ; 上料机构状态
; rung 14
LD=(300) 4011 &12  ; 上料机构状态
AND W19.10  ; 启动状态
OUT TR0
LDNOT T0086  ; 移栽前电池感应
ANDNOT T0087  ; 移栽后电池感应
ORNOT T0087  ; 移栽后电池感应
ANDLD
AND W20.00  ; 移栽伺服在上料位置
ANDNOT 2.10  ; 拉倒衔接处有料
LD H21.00  ; 移栽#1有料
ANDNOT H21.01  ; #1电池绝缘检测NG
ORNOT H21.00  ; 移栽#1有料
ANDLD
RSET W18.02  ; 上料阻挡气缸伸出
LD TR0
AND T0000  ; 上料阻挡气缸缩回位时间
ANDNOT 0.01  ; 上料有料感应
TIMX(550) 0294 &8  ; 来料流出时间
AND T0294  ; 来料流出时间
OUT TR0
AND P_Off
RSTA(531) H18 &2 &2  ; 上料电池的检测结果
LD TR0
@SET H18.00  ; 扫码OK
@SET H18.04  ; 进料到移栽位有料
MOV(021) &1 4011  ; 上料机构状态

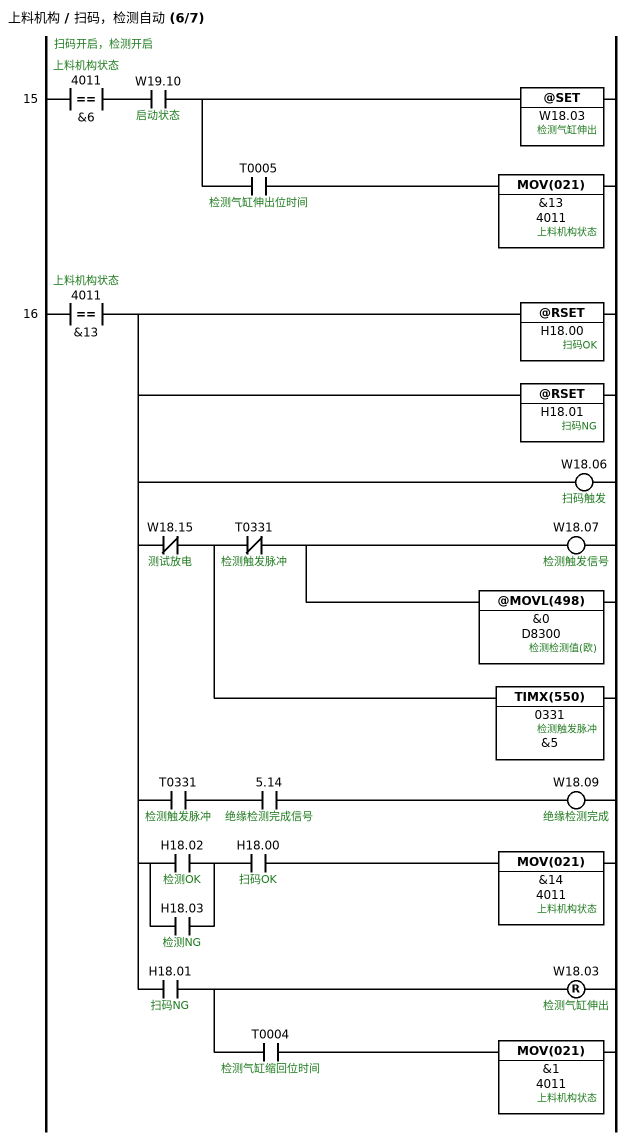
; rung 15: 扫码开启，检测开启
LD=(300) 4011 &6  ; 上料机构状态
AND W19.10  ; 启动状态
@SET W18.03  ; 检测气缸伸出
AND T0005  ; 检测气缸伸出位时间
MOV(021) &13 4011  ; 上料机构状态
; rung 16
LD=(300) 4011 &13  ; 上料机构状态
OUT TR0
@RSET H18.00  ; 扫码OK
@RSET H18.01  ; 扫码NG
OUT W18.06  ; 扫码触发
ANDNOT W18.15  ; 测试放电
OUT TR1
ANDNOT T0331  ; 检测触发脉冲
OUT W18.07  ; 检测触发信号
@MOVL(498) &0 D8300  ; 检测检测值(欧)
LD TR1
TIMX(550) 0331 &5  ; 检测触发脉冲
LD TR0
AND T0331  ; 检测触发脉冲
AND 5.14  ; 绝缘检测完成信号
OUT W18.09  ; 绝缘检测完成
LD TR0
LD H18.02  ; 检测OK
OR H18.03  ; 检测NG
ANDLD
AND H18.00  ; 扫码OK
MOV(021) &14 4011  ; 上料机构状态
LD TR0
AND H18.01  ; 扫码NG
RSET W18.03  ; 检测气缸伸出
AND T0004  ; 检测气缸缩回位时间
MOV(021) &1 4011  ; 上料机构状态

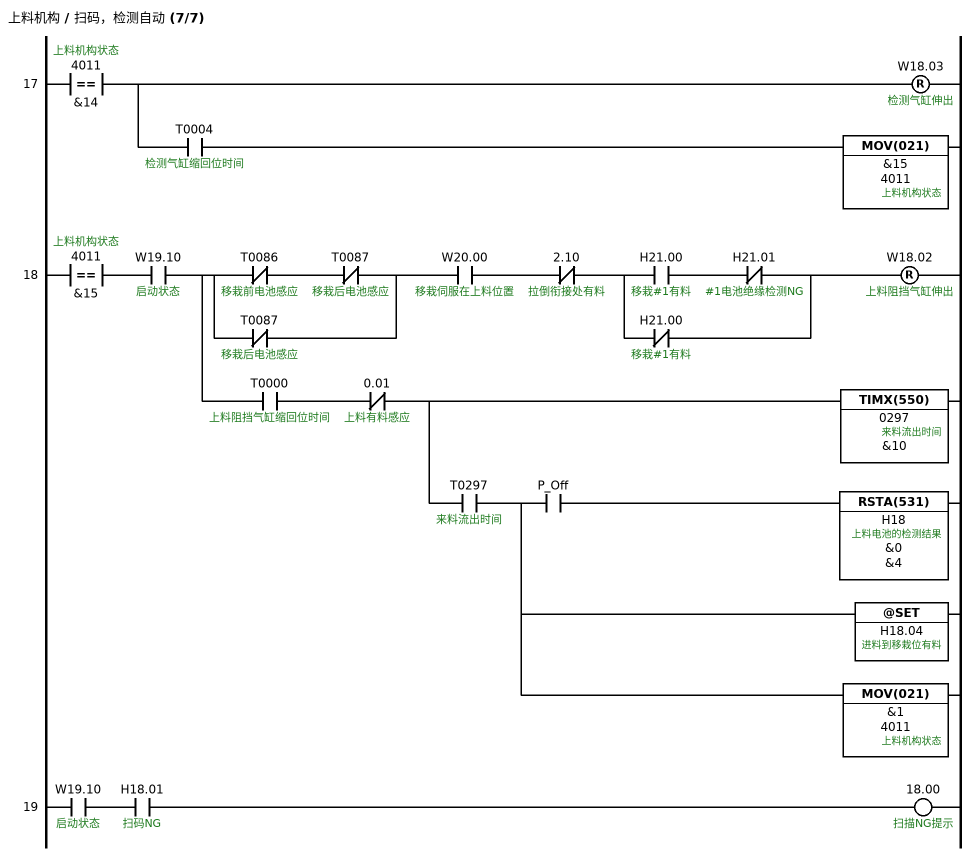
; rung 17
LD=(300) 4011 &14  ; 上料机构状态
RSET W18.03  ; 检测气缸伸出
AND T0004  ; 检测气缸缩回位时间
MOV(021) &15 4011  ; 上料机构状态
; rung 18
LD=(300) 4011 &15  ; 上料机构状态
AND W19.10  ; 启动状态
OUT TR0
LDNOT T0086  ; 移栽前电池感应
ANDNOT T0087  ; 移栽后电池感应
ORNOT T0087  ; 移栽后电池感应
ANDLD
AND W20.00  ; 移栽伺服在上料位置
ANDNOT 2.10  ; 拉倒衔接处有料
LD H21.00  ; 移栽#1有料
ANDNOT H21.01  ; #1电池绝缘检测NG
ORNOT H21.00  ; 移栽#1有料
ANDLD
RSET W18.02  ; 上料阻挡气缸伸出
LD TR0
AND T0000  ; 上料阻挡气缸缩回位时间
ANDNOT 0.01  ; 上料有料感应
TIMX(550) 0297 &10  ; 来料流出时间
AND T0297  ; 来料流出时间
OUT TR0
AND P_Off
RSTA(531) H18 &0 &4  ; 上料电池的检测结果
LD TR0
@SET H18.04  ; 进料到移栽位有料
MOV(021) &1 4011  ; 上料机构状态
; rung 19
LD W19.10  ; 启动状态
AND H18.01  ; 扫码NG
OUT 18.00  ; 扫描NG提示

### Section 扫描

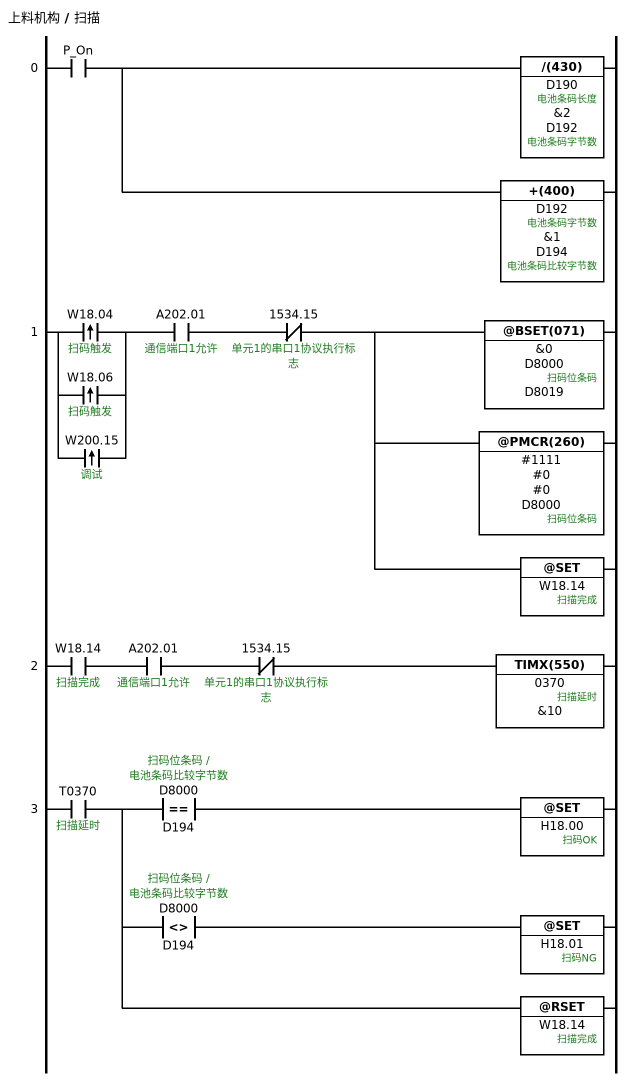
; rung 0
LD P_On
/(430) D190 &2 D192  ; 电池条码长度, 电池条码字节数
+(400) D192 &1 D194  ; 电池条码字节数, 电池条码比较字节数
; rung 1
@LD W18.04  ; 扫码触发
@OR W18.06  ; 扫码触发
@OR W200.15  ; 调试
AND A202.01  ; 通信端口1允许
ANDNOT 1534.15  ; 单元1的串口1协议执行标志
@BSET(071) &0 D8000 D8019  ; 扫码位条码
@PMCR(260) #1111 #0 #0 D8000  ; 扫码位条码
@SET W18.14  ; 扫描完成
; rung 2
LD W18.14  ; 扫描完成
AND A202.01  ; 通信端口1允许
ANDNOT 1534.15  ; 单元1的串口1协议执行标志
TIMX(550) 0370 &10  ; 扫描延时
; rung 3
LD T0370  ; 扫描延时
OUT TR0
AND=(300) D8000 D194  ; 扫码位条码, 电池条码比较字节数
@SET H18.00  ; 扫码OK
LD TR0
AND<>(305) D8000 D194  ; 扫码位条码, 电池条码比较字节数
@SET H18.01  ; 扫码NG
LD TR0
@RSET W18.14  ; 扫描完成

### Section 外部输出

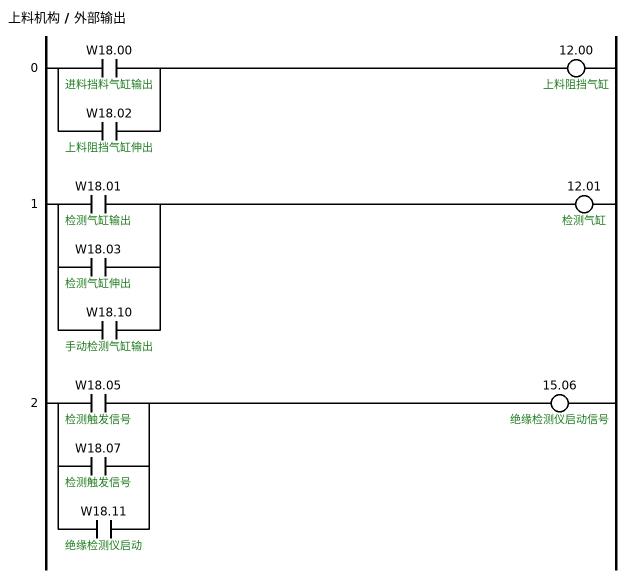
; rung 0
LD W18.00  ; 进料挡料气缸输出
OR W18.02  ; 上料阻挡气缸伸出
OUT 12.00  ; 上料阻挡气缸
; rung 1
LD W18.01  ; 检测气缸输出
OR W18.03  ; 检测气缸伸出
OR W18.10  ; 手动检测气缸输出
OUT 12.01  ; 检测气缸
; rung 2
LD W18.05  ; 检测触发信号
OR W18.07  ; 检测触发信号
OR W18.11  ; 绝缘检测仪启动
OUT 15.06  ; 绝缘检测仪启动信号

### Section 自动报警

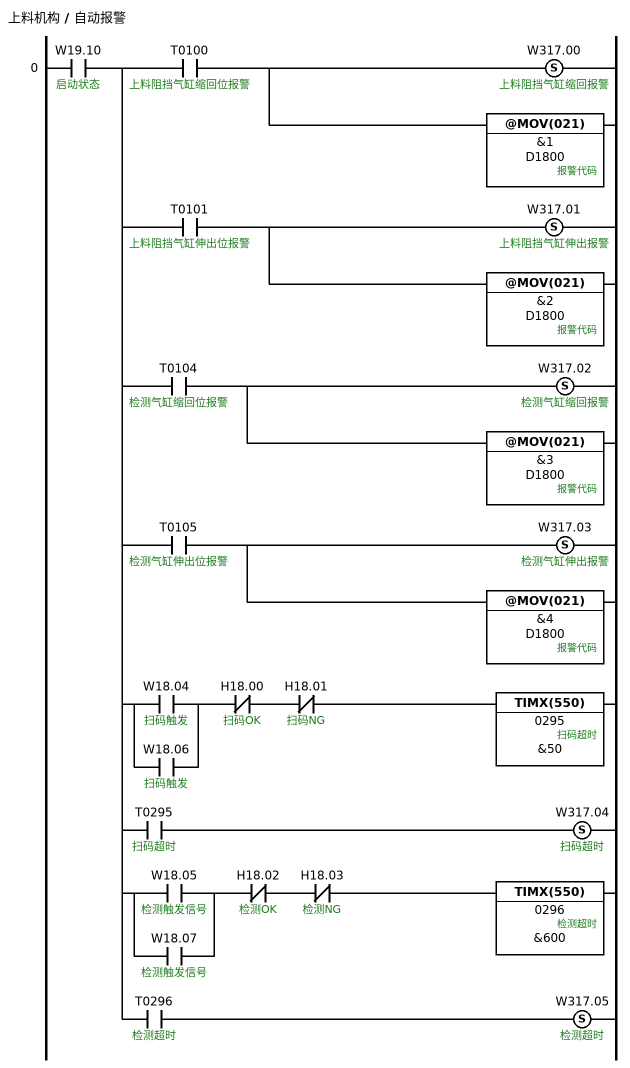
; rung 0
LD W19.10  ; 启动状态
OUT TR0
AND T0100  ; 上料阻挡气缸缩回位报警
SET W317.00  ; 上料阻挡气缸缩回报警
@MOV(021) &1 D1800  ; 报警代码
LD TR0
AND T0101  ; 上料阻挡气缸伸出位报警
SET W317.01  ; 上料阻挡气缸伸出报警
@MOV(021) &2 D1800  ; 报警代码
LD TR0
AND T0104  ; 检测气缸缩回位报警
SET W317.02  ; 检测气缸缩回报警
@MOV(021) &3 D1800  ; 报警代码
LD TR0
AND T0105  ; 检测气缸伸出位报警
SET W317.03  ; 检测气缸伸出报警
@MOV(021) &4 D1800  ; 报警代码
LD TR0
LD W18.04  ; 扫码触发
OR W18.06  ; 扫码触发
ANDLD
ANDNOT H18.00  ; 扫码OK
ANDNOT H18.01  ; 扫码NG
TIMX(550) 0295 &50  ; 扫码超时
LD TR0
AND T0295  ; 扫码超时
SET W317.04  ; 扫码超时
LD TR0
LD W18.05  ; 检测触发信号
OR W18.07  ; 检测触发信号
ANDLD
ANDNOT H18.02  ; 检测OK
ANDNOT H18.03  ; 检测NG
TIMX(550) 0296 &600  ; 检测超时
LD TR0
AND T0296  ; 检测超时
SET W317.05  ; 检测超时

### Section 复位

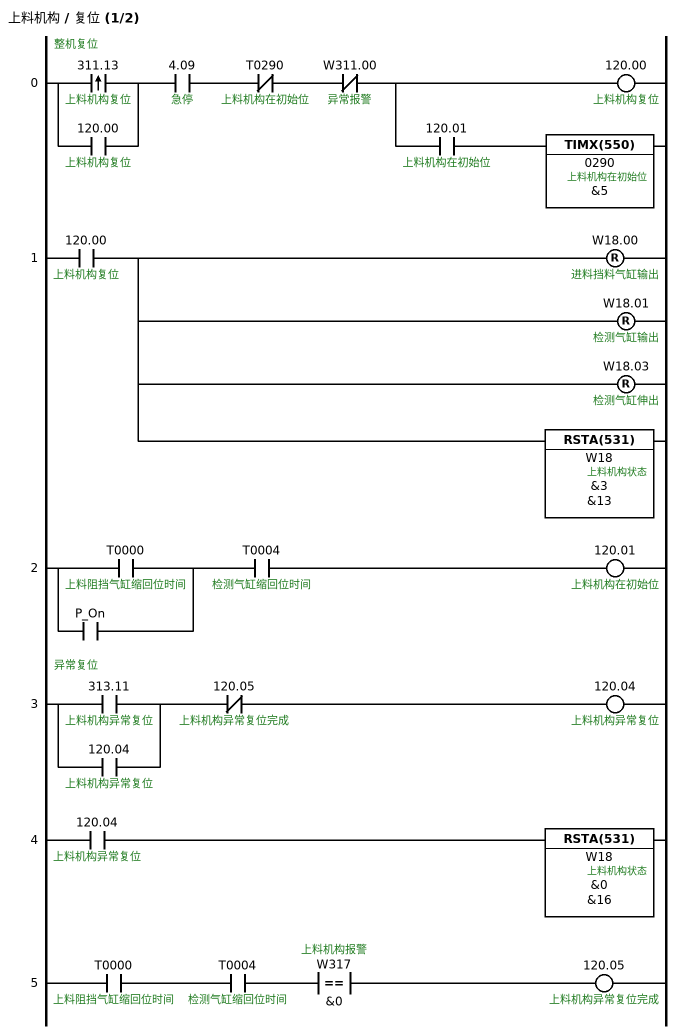
; rung 0: 整机复位
@LD 311.13  ; 上料机构复位
OR 120.00  ; 上料机构复位
AND 4.09  ; 急停
ANDNOT T0290  ; 上料机构在初始位
ANDNOT W311.00  ; 异常报警
OUT 120.00  ; 上料机构复位
AND 120.01  ; 上料机构在初始位
TIMX(550) 0290 &5  ; 上料机构在初始位
; rung 1
LD 120.00  ; 上料机构复位
RSET W18.00  ; 进料挡料气缸输出
RSET W18.01  ; 检测气缸输出
RSET W18.03  ; 检测气缸伸出
RSTA(531) W18 &3 &13  ; 上料机构状态
; rung 2
LD T0000  ; 上料阻挡气缸缩回位时间
OR P_On
AND T0004  ; 检测气缸缩回位时间
OUT 120.01  ; 上料机构在初始位
; rung 3: 异常复位
LD 313.11  ; 上料机构异常复位
OR 120.04  ; 上料机构异常复位
ANDNOT 120.05  ; 上料机构异常复位完成
OUT 120.04  ; 上料机构异常复位
; rung 4
LD 120.04  ; 上料机构异常复位
RSTA(531) W18 &0 &16  ; 上料机构状态
; rung 5
LD T0000  ; 上料阻挡气缸缩回位时间
AND T0004  ; 检测气缸缩回位时间
AND=(300) W317 &0  ; 上料机构报警
OUT 120.05  ; 上料机构异常复位完成

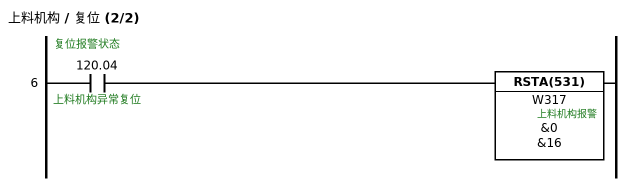
; rung 6: 复位报警状态
LD 120.04  ; 上料机构异常复位
RSTA(531) W317 &0 &16  ; 上料机构报警

### Section END
; rung 0
END(001)

## Program 上料移栽 (cyclic task 3)

### Section 上料移栽手动

